PROGRAM MAIN
VAR
    
END_VAR

RunStudent();

END_PROGRAM

(* stored: Version 1.1.0.1
   POU MAIN: Id {c85ca7f7-62e4-4195-a50a-ed021ea2dff4}, SpecialFunc None *)
